INTERFACE IVisitor

PROPERTY ActualValue : REAL
GET
END_GET
END_PROPERTY

METHOD updateValue : REAL
VAR_INPUT
	value: REAL;
END_VAR
END_METHOD

END_INTERFACE

(* stored: Version 1.1.0.1
   Itf IVisitor: Id {3c58ef9c-7e84-4c2f-bd79-93b71c257255}
   Property ActualValue: Id {6ba75df2-8cb7-4218-879b-f0d43aaffe03}
   Get Get: Id {8507bf57-0be5-4ac1-a8dc-7bcc936f819b}
   Method updateValue: Id {4fd80157-8a5d-43ed-8375-3336bfc32f7b} *)
